DEVICE_TYPE RMT_FLASHER (* Remote FLASHER4 Server *)
  (* Standard: 61499-1 *)
  (* Version 0.0, 2006-10-27, JHC, Holobloc Inc, Derived from FLASHER_TESTR *)
  (* Compiler header: package fb.rt.doc; *)
  (* Compiler classdef: public class RMT_FLASHER extends RMT_DEV *)
  (* Compiler Java Sun JDK 1.5.0 *)
  RESOURCE RES1 : EMB_RES
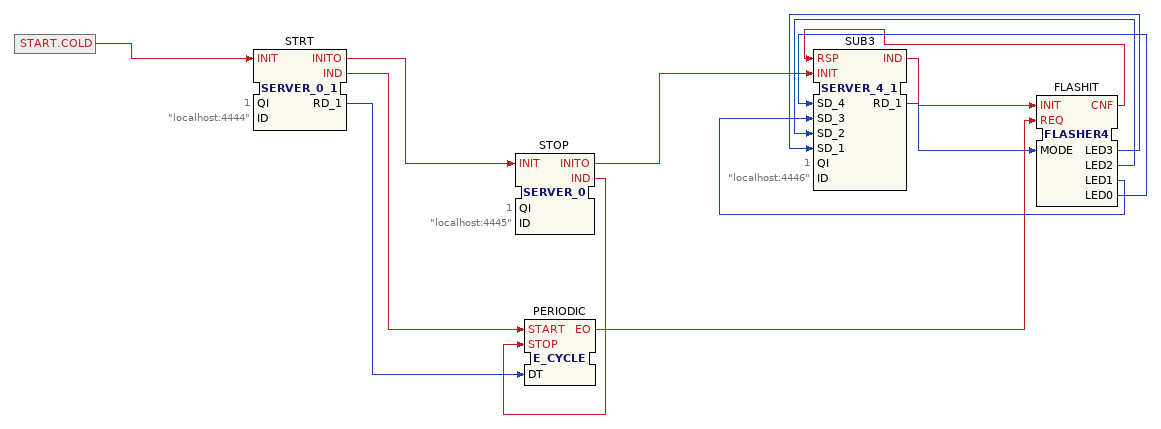
    FBS
      SUB3 : SERVER_4_1(QI := 1, ID := "localhost:4446");
      PERIODIC : E_CYCLE;
      FLASHIT : FLASHER4;
      STRT : SERVER_0_1(QI := 1, ID := "localhost:4444");
      STOP : SERVER_0(QI := 1, ID := "localhost:4445");
    END_FBS
    EVENT_CONNECTIONS
      SUB3.IND TO FLASHIT.INIT;
      PERIODIC.EO TO FLASHIT.REQ;
      FLASHIT.CNF TO SUB3.RSP;
      START.COLD TO STRT.INIT;
      STRT.INITO TO STOP.INIT;
      STRT.IND TO PERIODIC.START;
      STOP.INITO TO SUB3.INIT;
      STOP.IND TO PERIODIC.STOP;
    END_CONNECTIONS
    DATA_CONNECTIONS
      FLASHIT.LED0 TO SUB3.SD_4;
      FLASHIT.LED1 TO SUB3.SD_3;
      FLASHIT.LED2 TO SUB3.SD_2;
      FLASHIT.LED3 TO SUB3.SD_1;
      SUB3.RD_1 TO FLASHIT.MODE;
      STRT.RD_1 TO PERIODIC.DT;
    END_CONNECTIONS
  END_RESOURCE
END_DEVICE_TYPE
